// TIA Portal project "3M3" (V16)

(* hardware
DEVICE "S7-1200 station_1"  S7-1200 Station
   slot 0: "Rack_0"  S7-1200 Rack  Rack  V1.0
   slot 1: "PLC_1"  CPU 1212C AC/DC/Rly  6ES7 212-1BE40-0XB0  V4.4
*)

// ===== PLC "PLC_1"  CPU 1212C AC/DC/Rly =====

VAR_GLOBAL   // PLC tag table "Default tag table"
   "START" AT %I0.1 : Bool;
   "MOTOR1" AT %Q0.0 : Bool;
   "MOTOR2" AT %Q0.1 : Bool;
   "MOTOR3" AT %Q0.2 : Bool;
   "Tag_1" AT %M0.0 : Bool;
   "Tag_2" AT %M0.1 : Bool;
   "Tag_3" AT %M0.3 : Bool;
   "Tag_4" AT %M0.4 : Bool;
   "Tag_5" AT %M0.5 : Bool;
END_VAR

// folder: System blocks/Program resources

DATA_BLOCK "COUNTER"   // DB1
{ S7_Optimized_Access := 'TRUE' }
AUTHOR : Simatic
FAMILY : IEC
NAME : CNTR
VERSION : 1.0
// stored: InstanceOfName IEC_COUNTER
"IEC_COUNTER"
BEGIN
END_DATA_BLOCK

// folder: (top level)

ORGANIZATION_BLOCK "Main"   // OB1, LAD, ProgramCycle
TITLE = "Main Program Sweep (Cycle)"
{ S7_Optimized_Access := 'TRUE' }
VERSION : 0.1
   VAR_INPUT
      Initial_Call : Bool;   // Initial call of this OB
      Remanence : Bool;   // =True, if remanent data are available
   END_VAR
   VAR_TEMP   // added for the SCL form of the ladder/FBD networks
      _w1 : Bool;
   END_VAR
BEGIN

REGION Network 1
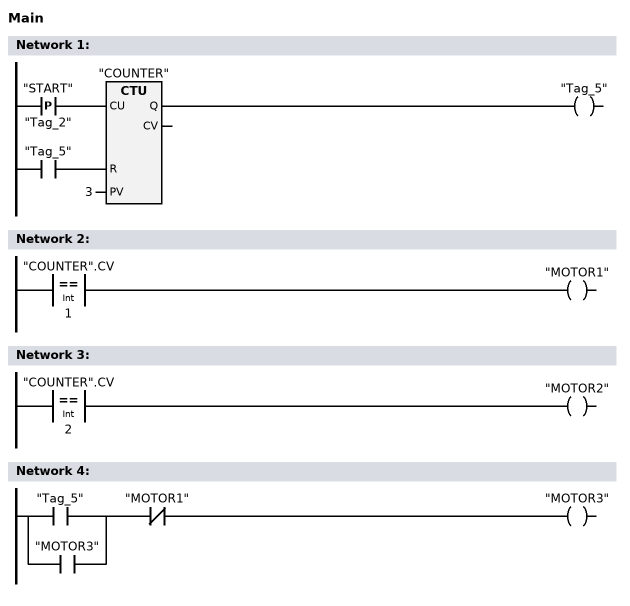
   #_w1 := "START" AND NOT "Tag_2";   // rising edge of "START"
   "Tag_2" := "START";
   "COUNTER".CTU(CU := #_w1, R := "Tag_5", PV := 3);
   "Tag_5" := "COUNTER".Q;
END_REGION

REGION Network 2
   RUNG wire#powerrail
      { S7_Templates := "SrcType := Int" } EQ_Contact(in1 := "COUNTER".CV, in2 := 1)
      Coil( "MOTOR1" )
   END_RUNG
   // the same network as SCL:
   "MOTOR1" := "COUNTER".CV = 1;
END_REGION

REGION Network 3
   RUNG wire#powerrail
      { S7_Templates := "SrcType := Int" } EQ_Contact(in1 := "COUNTER".CV, in2 := 2)
      Coil( "MOTOR2" )
   END_RUNG
   // the same network as SCL:
   "MOTOR2" := "COUNTER".CV = 2;
END_REGION

REGION Network 4
   RUNG wire#powerrail
      Contact( "Tag_5" )
      wire#w1
      I_Contact( "MOTOR1" )
      Coil( "MOTOR3" )
   END_RUNG
   RUNG wire#powerrail
      Contact( "MOTOR3" )
   END_RUNG wire#w1
   // the same network as SCL:
   "MOTOR3" := ("Tag_5" OR "MOTOR3") AND NOT "MOTOR1";
END_REGION
END_ORGANIZATION_BLOCK